PROGRAM UDPTest
VAR
	socketCreate:	FB_SocketUdpCreate;
	socketSend:		FB_SocketUdpSendTo;
	createNow: 		BOOL;
	sendNow:		BOOL;
	sMsg:			STRING[20] := 'Hello World';
	configCreate: 	BOOL := true;
	configSend: 	BOOL := TRUE;
END_VAR




IF configCreate THEN
	socketCreate.sSrvNetId := '';
	socketCreate.sLocalHost := '127.0.0.1';
	socketCreate.nLocalPort := 52123;
	socketCreate.tTimeout := T#5S;
	configCreate := FALSE;
END_IF


//IF createNow THEN
	socketCreate.bExecute := createNow;
//	createNow := FALSE;
//END_IF

IF configSend THEN
	socketSend.sSrvNetId := '';
	socketSend.sRemoteHost := '127.0.0.1';
	socketSend.nRemotePort := 8000;
	socketSend.cbLen := INT_TO_UDINT(LEN(sMsg));
	socketSend.pSrc := ADR(sMsg);
	socketSend.tTimeout := T#5S;
	configSend := FALSE;
END_IF

socketSend.hSocket := socketCreate.hSocket;

socketSend.bExecute := sendNow;
sendNow := FALSE;

// Call fbs
socketCreate();
socketSend();

END_PROGRAM

(* stored: Version 1.1.0.1, ProductVersion 3.1.4024.12
   POU UDPTest: Id {d4ea590e-d88c-4479-a1c6-26e991dfdda3}, SpecialFunc None *)
